// TIA Portal V17 export
// export: Created 2025-06-26T06:49:29.7577471Z, ExportSetting WithDefaults, DisplayName Totally Integrated Automation Portal, DisplayVersion V17 Update 8, DisplayName TIA Portal Openness, DisplayVersion V17 Update 8, DisplayName TIA Portal Version Control Interface, DisplayVersion V17, DisplayName STEP 7 Professional, DisplayVersion V17 Update 8, DisplayName STEP 7 Safety, DisplayVersion V17 Update 6, DisplayName WinCC Advanced, DisplayVersion V17 Update 8
TYPE "stHeartbeat"
// stored: IsFailsafeCompliant false
   STRUCT
      bOut : Bool;   // Bit sent to remote partner
      bIn : Bool;   // Bit received from remote partner
      bEnable : Bool;   // 1 = run heartbeat, 0 = disabled
      bOk : Bool;   // 1 = heatbeat ok, 0 = timeout
      nState : USInt;   // Heartbeat state
      tTimeout : Time;   // Timeout before comm error
   END_STRUCT;
END_TYPE
